FUNCTION_BLOCK FB_RecipeBuilderWings EXTENDS FB_PackML_BaseModule IMPLEMENTS I_RecipeBuilder

VAR
	RecipeBuilder_HMI: ST_RecipeBuilder_HMI;
	_Config					:ST_RecipeBuilder_Config;
	_PanelFrontLength		:REAL;  
	_PanelFrontWidth		:REAL;      
	_PanelHeight			:REAL;    
	_RailHeightCorrection	:REAL;
END_VAR

METHOD Build : BOOL
VAR_INPUT
	PanelWidth	: REAL;
	PanelLength	: REAL;
	PanelHeight	: REAL;
	CuttingOverpass	: REAL;
	RailHeightCorrection	: REAL;
END_VAR
END_METHOD

PROPERTY Config : ST_RecipeBuilder_Config
GET
Config := _Config;
END_GET
SET
RecipeBuilder_HMI.Config := Config;
END_SET
END_PROPERTY

// Provides interlocks for HMI control and updates HMI status information for this module
METHOD PROTECTED HMICommunication

// This method is called cyclically by CyclicLogic()
_PanelFrontWidth      := RecipeBuilder_HMI.Config.PanelFrontWidht;
_PanelFrontLength     := RecipeBuilder_HMI.Config.PanelFrontLength;
_PanelHeight          := RecipeBuilder_HMI.Config.PanelHeight;
_RailHeightCorrection := RecipeBuilder_HMI.Config.RailHeightCorrection;
END_METHOD

PROPERTY SegmentsCutX : ARRAY [1..32] OF ST_CutSegment
GET
END_GET
END_PROPERTY

PROPERTY SegmentsCutY : ARRAY [1..32] OF ST_CutSegment
GET
END_GET
END_PROPERTY


PROPERTY SegmentsGroove : ARRAY [1..32] OF ST_CutSegment
GET
END_GET
END_PROPERTY


PROPERTY SegmentsToCutX : INT
GET
END_GET
END_PROPERTY


PROPERTY SegmentsToCutY : INT
GET
END_GET
END_PROPERTY


PROPERTY SegmentsToGroove : INT
GET
END_GET
END_PROPERTY

END_FUNCTION_BLOCK

(* stored: Version 1.1.0.1, ProductVersion 3.1.4024.15
   POU FB_RecipeBuilderWings: Id {3f83a514-1f2f-4e3d-921c-ca7c0b60e17f}, SpecialFunc None
   Method Build: Id {c08ade7c-db75-4c50-8457-5bb392619adf}
   Property Config: Id {e53be9fd-6b88-49c9-8736-ae6ec54e43d8}
   Get Get: Id {0bd9a01b-52a6-47dd-b6fc-d6ccf0a489a9}
   Set Set: Id {e2eb298e-f304-4e9d-ab04-77a183356e49}
   Method HMICommunication: Id {5b58a0e6-30db-439b-a833-a33f4b223005}
   Property SegmentsCutX: Id {9152e646-9866-44c9-b9e6-5a764990d7d4}
   Get Get: Id {8272f94b-fbfa-4156-a332-efb73ed5cf2e}
   Property SegmentsCutY: Id {255ca92b-c547-401c-9784-b32df54e5e2a}
   Get Get: Id {4b559848-f1de-4c18-834d-4d2909a2699d}
   Property SegmentsGroove: Id {a6cc8c84-07e4-4531-824b-69c46a3f14a3}
   Get Get: Id {7a846cca-77b5-4d85-b851-6d33d3df4235}
   Property SegmentsToCutX: Id {e45efa5d-ccfc-458e-9811-5f080acfb1d1}
   Get Get: Id {58e9fc3c-a2ea-47ff-862f-fb085769cffc}
   Property SegmentsToCutY: Id {0f05ab0b-f50d-4ba7-9a3d-ced7155bbd03}
   Get Get: Id {dd01e30b-5156-462c-981f-e1777bde948b}
   Property SegmentsToGroove: Id {e4a3954d-3a1b-4d86-a891-2e859afd79f8}
   Get Get: Id {166af98c-be7e-4a9c-8000-ac82596ec13a} *)
